FUNCTION_BLOCK FB_Test_Base_Not EXTENDS FB_UnitTestBase
VAR_INPUT
END_VAR
VAR_OUTPUT
END_VAR
VAR
END_VAR

(******************************************************************************
Baustein: FB_Test_Base_Not.cleanup
Spezifikation: doc/Spezifikation.pdf, Kap. x.y.z
-------------------------------------------------------------------------------
erstellt:
von:
Geändert:
von:
-------------------------------------------------------------------------------
Beschreibung
Diese Methode...

-------------------------------------------------------------------------------
Input
-

Output
-
******************************************************************************)
METHOD PUBLIC cleanup : BOOL
VAR_INPUT
END_VAR

	cleanup := true;
END_METHOD

(******************************************************************************
Baustein: FB_Test_Base_Not.execute
Spezifikation: doc/Spezifikation.pdf, Kap. x.y.z
-------------------------------------------------------------------------------
erstellt:
von:
Geändert:
von:
-------------------------------------------------------------------------------
Beschreibung
Diese Methode...

-------------------------------------------------------------------------------
Input
-

Output
-
******************************************************************************)
METHOD PUBLIC execute : BOOL
VAR_INPUT
END_VAR
VAR
	bValue1   : ARRAY[0..10] OF BOOL;
	bValue2   : ARRAY[0..10] OF BOOL;
	s8Value1  : ARRAY[0..10] OF SINT;
	s8Value2  : ARRAY[0..10] OF SINT;
	u8Value1  : ARRAY[0..10] OF USINT;
	u8Value2  : ARRAY[0..10] OF USINT;	
	s16Value1 : ARRAY[0..10] OF INT;
	s16Value2 : ARRAY[0..10] OF INT;
	u16Value1 : ARRAY[0..10] OF UINT;
	u16Value2 : ARRAY[0..10] OF UINT;		
	s32Value1 : ARRAY[0..10] OF DINT;
	s32Value2 : ARRAY[0..10] OF DINT;
	u32Value1 : ARRAY[0..10] OF UDINT;
	u32Value2 : ARRAY[0..10] OF UDINT;	
	r32Value1 : ARRAY[0..10] OF REAL;
	r32Value2 : ARRAY[0..10] OF REAL;
	r64Value1 : ARRAY[0..10] OF LREAL;
	r64Value2 : ARRAY[0..10] OF LREAL;
END_VAR

	bValue1[0] := FALSE;
	bValue2[0] := TRUE;
	assertNotEQUAL(bValue1, bValue2);

	s8Value1[0] := 31;
	s8Value2[0] := 32;
	assertNotEQUAL(s32Value1, s32Value2);

	u8Value1[0] := 1;
	u8Value2[0] := 34;
	assertNotEQUAL(s32Value1, s32Value2);
	
	s16Value1[0] := 1323;
	s16Value2[0] := 4324;
	assertNotEQUAL(s32Value1, s32Value2);

	u16Value1[0] := 3124;
	u16Value2[0] := 4232;
	assertNotEQUAL(s32Value1, s32Value2);
	
	s32Value1[0] := 1244;
	s32Value2[0] := 1593;
	assertNotEQUAL(s32Value1, s32Value2);

	u32Value1[0] := 4344;
	u32Value2[0] := 3424;
	assertNotEQUAL(s32Value1, s32Value2);
	
	r32Value1[0] := 133.53245;
	r32Value2[0] := 5345.53245;
	assertNotEQUAL(r32Value1, r32Value2);

	r64Value1[0] := 1232.53325;
	r64Value2[0] := 1345.53325;
	assertNotEQUAL(r32Value1, r32Value2);
	
	execute := TRUE;
END_METHOD

(******************************************************************************
Baustein: FB_Test_Base_Not.prepare
Spezifikation: doc/Spezifikation.pdf, Kap. x.y.z
-------------------------------------------------------------------------------
erstellt:
von:
Geändert:
von:
-------------------------------------------------------------------------------
Beschreibung
Diese Methode...

-------------------------------------------------------------------------------
Input
-

Output
-
******************************************************************************)
METHOD PUBLIC prepare : BOOL
VAR_INPUT
END_VAR

	prepare := true;
END_METHOD

END_FUNCTION_BLOCK

(* stored: Version 1.1.0.1, ProductVersion 3.1.4024.3
   POU FB_Test_Base_Not: Id {fcf08a4b-84b3-4de6-9021-24a73f13f2bf}, SpecialFunc None
   Method cleanup: Id {65da6c5b-32cd-49b2-8efb-d7e2ddbdaf15}
   Method execute: Id {787a6e5e-98af-47ae-8dc1-33d98cab30ec}
   Method prepare: Id {6212eda2-4fb6-4cf5-a93a-1b3be7bda95e} *)
